FUNCTION_BLOCK MTCSChangeInstrumentProcess EXTENDS BaseProcess
VAR_INPUT
	///Arguments to be set, before writing do_request TRUE
	{attribute 'OPC.UA.DA' := '1'}
	set: MTCSChangeInstrumentProcessArgs;
END_VAR
VAR_OUTPUT
	///Arguments in use by the process, if do_request was accepted
	{attribute 'OPC.UA.DA' := '1'}
	{attribute 'OPC.UA.DA.Access' := '1'}
	get: MTCSChangeInstrumentProcessArgs;
END_VAR
VAR_IN_OUT
END_VAR
VAR
END_VAR

IF do_request THEN
    do_request_result := request( name := set.name );
    do_request := FALSE;
END_IF;
SUPER^();

{attribute 'TcRpcEnable' := '1'}
METHOD request : RequestResults
VAR_INPUT
	///Name of the instrument
	name: STRING;
END_VAR
VAR_OUTPUT
END_VAR
VAR_IN_OUT
END_VAR
VAR
END_VAR
IF THIS^.statuses.enabledStatus.enabled THEN
    THIS^.start( name := name );
    request := RequestResults.ACCEPTED;
ELSE
    request := RequestResults.REJECTED;
END_IF;
END_METHOD

{attribute 'TcRpcEnable' := '1'}
METHOD start
VAR_INPUT
	///Name of the instrument
	name: STRING;
END_VAR
VAR_OUTPUT
END_VAR
VAR_IN_OUT
END_VAR
VAR
END_VAR
THIS^.get.name := name;
THIS^.statuses.busyStatus( isBusy := TRUE );
THIS^.statuses.healthStatus( isGood := TRUE );
END_METHOD

END_FUNCTION_BLOCK

(* stored: Version 1.1.0.1, ProductVersion 3.1.4019.2
   POU MTCSChangeInstrumentProcess: Id {0b716df1-dbb3-4f32-8c3d-e523aa1fdefa}, SpecialFunc None
   Method request: Id {260166e5-b28d-4f0a-b68c-493772672eb6}
   Method start: Id {e4ac2390-6bde-4403-b685-57c942550184} *)
